// TIA Portal V19 export
TYPE "actionEmManager"
// stored: Namespace Unit2
   STRUCT
      emCommand { ExternalAccessible := 'False'; ExternalVisible := 'False'; ExternalWritable := 'False'} : "LUC_typeStateCommands";
      emStatus { ExternalAccessible := 'False'; ExternalVisible := 'False'; ExternalWritable := 'False'} : "LUC_typeStates";
   END_STRUCT;
END_TYPE
